(* CODESYS project mobject-enumerable.library
   Company: mobject
   DefaultNamespace: mobject-enumerable
   Version: 1.2.0
   Placeholder: mobject-enumerable
   Author: mobject dev team
   Title: mobject-enumerable

Project tree, tasks and I/O mapping:
  libraries: mobject-disposable, 1.1.1 (mobject); Tc2_System, * (Beckhoff Automation GmbH)
  Interfaces/
    Enumerators/
      interface I_ForwardEnumerator: IsValid, MoveNext, Reset, TryGet, TryGetTo
      interface I_KeyValueForwardEnumerator: Key
    interface I_Enumerable: GetEnumerator
    interface I_KeyValueEnumerable: GetKeyValueEnumerator
*)

// Interfaces/Enumerators/I_ForwardEnumerator
INTERFACE I_ForwardEnumerator EXTENDS I_Disposable

PROPERTY PUBLIC IsValid : BOOL
GET
END_GET
END_PROPERTY

METHOD PUBLIC MoveNext : BOOL
END_METHOD

METHOD PUBLIC Reset
END_METHOD

METHOD PUBLIC TryGet : BOOL;
VAR_INPUT
    Destination : ANY;
END_VAR
END_METHOD

METHOD PUBLIC TryGetTo : BOOL;
VAR_INPUT
    DestinationAddress : PVOID;
    DestinationSize : UDINT;
END_VAR
END_METHOD

END_INTERFACE

// Interfaces/Enumerators/I_KeyValueForwardEnumerator
INTERFACE I_KeyValueForwardEnumerator EXTENDS I_ForwardEnumerator

PROPERTY Key : T_MAXSTRING
GET
END_GET
END_PROPERTY

END_INTERFACE

// Interfaces/I_Enumerable
INTERFACE I_Enumerable EXTENDS __SYSTEM.IQueryInterface

METHOD PUBLIC GetEnumerator : I_ForwardEnumerator
END_METHOD

END_INTERFACE

// Interfaces/I_KeyValueEnumerable
INTERFACE I_KeyValueEnumerable EXTENDS __SYSTEM.IQueryInterface

METHOD PUBLIC GetKeyValueEnumerator : I_KeyValueForwardEnumerator
END_METHOD

END_INTERFACE
